{attribute 'GeneratedUsingTerminal: EQ2008-0002-0016'}
{attribute addProperty BoxType "EQ2008-0002-0016"}
{attribute addProperty Id "WcStateAT %I*BOOL1"}
{attribute addProperty CRC "187373305"}
{attribute addProperty Size "1"}
TYPE WcState_0B2B16F9 :
STRUCT
	{attribute addProperty Name "WcState"}
	WcState AT %I* : BOOL;
END_STRUCT
END_TYPE

(* stored: Version 1.2.0.0, ProductVersion 3.1.4024.9
   DUT WcState_0B2B16F9: Id {8a967518-0b78-4003-97c6-d54de7fa3cd8} *)
